{attribute 'qualified_only'}
{attribute 'strict'}
TYPE BessStateControl :
(
	STOP := 2,
	RUN := 6
)UINT;
END_TYPE

(* stored: Version 1.1.0.1, ProductVersion 3.1.4024.11
   DUT BessStateControl: Id {b5cc1a4f-abd5-4f48-9485-4f66f8a21a26} *)
